(* IEC 61131-3 sources: teller/JD_Teller_LC2_V11/Class/WisComment, 1 file *)

(* ---- WisComment.st ---- *)
(*!
<Class
	Name               = "WisComment"
	Revision           = "1.0"
	RealtimeTask       = "false"
	CyclicTask         = "false"
	BackgroundTask     = "false"
	Sigmatek           = "false"
	OSInterface        = "false"
	HighPriority       = "false"
	Automatic          = "false"
	UpdateMode         = "Prescan"
	SharedCommandTable = "true"
	Objectsize         = "(284,120)">
	<Channels>
		<Server Name="Wis" Visualized="true" Initialize="false" WriteProtected="false" Retentive="false"/>
		<Client Name="ExtFilter" Required="true" Internal="false"/>
		<Client Name="String2" Required="true" Internal="true"/>
		<Client Name="System" Required="false" Internal="false"/>
	</Channels>
	<RevDoku>
		<Owner Company="JV" Author="JvD"/>
		<Dokumentation Revision="1.0" Date="2012-10-11" Author="JvD" Company="JV" Description="StringRam aan Client toegevoegd"/>
	</RevDoku>
	<Network Name="WisComment">
		<!-- List of Components in this network -->
		<Components>
			<Object
				Name       = "String2"
				Class      = "String"
				Position   = "(240,270)"
				Visualized = "true">
				<Channels>
					<Server Name="Data"/>
					<Client Name="SingleRealloc" Value="1"/>
				</Channels>
			</Object>
		</Components>
		<Comments>
		</Comments>
		<!-- List of Connections in this network -->
		<Connections>
			<Connection Source="this.String2" Destination="String2.Data"/>
		</Connections>
		<!-- Headerfiles -->
		<Options>
		</Options>
	</Network>
</Class>
*)
WisComment : CLASS
  //Servers:
	Wis 	: SvrChCmd_DINT;
  //Clients:
	String2 	: CltChCmd_String;
	ExtFilter 	: CltChCmd_StringRAM;
	System 	: CltChCmd_System;
  //Variables:
  //Functions:

	FUNCTION VIRTUAL GLOBAL Init;

	FUNCTION VIRTUAL GLOBAL Wis::Write
		VAR_INPUT
			input (EAX) 	: DINT;
		END_VAR
		VAR_OUTPUT
			result (EAX) 	: DINT;
		END_VAR;
  //Tables:
	FUNCTION @STD
		VAR_OUTPUT
			ret_code	: CONFSTATES;
		END_VAR;
	FUNCTION GLOBAL TAB @CT_;
END_CLASS;

#pragma using String
#pragma usingLtd StringRAM
#pragma usingLtd System

FUNCTION VIRTUAL GLOBAL WisComment::Init

  String2.InitFromTable(udLen:= 0 , pData:= "");

END_FUNCTION

FUNCTION VIRTUAL GLOBAL WisComment::Wis::Write
	VAR_INPUT
		input (EAX) 	: DINT;
	END_VAR
	VAR_OUTPUT
		result (EAX) 	: DINT;
	END_VAR

	Wis := input;

  ExtFilter.WriteDataOff(udLen := 0, udOff := 0, pData := "");

 	result := Wis;

END_FUNCTION
